Yaskawa INFORM job: SKRZYNIA_4040_0_STOPNI_1OBR.JBI

/JOB
//NAME SKRZYNIA_4040_0_STOPNI_1OBR
///FOLDERNAME 02-SKRZYNIE_JOBS
//POS
///NPOS 413,413,0,35,0,0
///TOOL 0
///POSTYPE PULSE
///PULSE
C00000=1055,-24125,84372,288,19725,204
C00001=1055,-24125,84372,288,19725,204
C00002=0,-15438,65714,0,-68532,0
C00003=25524,-25821,36823,19654,-58495,38520
C00004=23988,-24960,37134,18595,-57837,38812
C00005=22822,-23954,37534,17811,-57199,39017
C00006=22935,-24057,37491,17887,-57262,38997
C00007=20006,-24258,37408,15644,-56932,39751
C00008=24402,-25289,37013,18874,-58060,38740
C00009=22585,-24665,40358,17164,-59622,30036
C00010=23477,-23257,40205,18030,-58646,29630
C00011=22519,-22398,40568,17384,-58125,29795
C00012=22700,-22567,40495,17506,-58225,29764
C00013=19339,-22794,40398,14955,-57865,30607
C00014=24825,-24328,39798,18931,-59350,29401
C00015=32755,-32613,25711,29640,-48730,33694
C00016=25632,-30899,26166,23992,-46203,35378
C00017=24264,-29862,26497,22996,-45413,35639
C00018=24403,-29974,26459,23097,-45496,35612
C00019=20575,-30233,26374,19602,-44891,36810
C00020=26556,-31526,25988,24663,-46720,35206
C00021=31152,-34007,25432,27964,-49085,34371
C00022=14779,-22420,82153,5620,-31515,42478
C00023=14779,-22420,82153,5620,-31515,42478
C00024=27667,-31817,30876,40298,-29340,25942
C00025=30467,-34548,18624,42252,-31099,25545
C00026=27667,-31817,21023,40298,-29340,25942
C00027=26226,-30681,21430,39338,-28403,26129
C00028=26403,-30829,21375,39455,-28520,26106
C00029=23300,-31093,21277,35654,-27590,27434
C00030=27667,-31817,21023,40298,-29340,25942
C00031=33767,-35384,20030,44426,-32984,25136
C00032=17528,-33021,25719,14295,-44761,40001
C00033=28412,-21339,35361,20830,-70681,36412
C00034=27333,-20260,35973,20228,-70115,36596
C00035=27399,-20329,35933,20265,-70150,36584
C00036=24360,-20684,35731,18412,-69734,37326
C00037=28877,-18893,40191,20941,-72149,36569
C00038=27817,-32566,25782,25532,-47502,36865
C00039=25779,-31294,26110,24054,-46400,37243
C00040=24344,-30243,26427,23007,-45578,37515
C00041=24432,-30312,26405,23072,-45630,37498
C00042=20021,-30599,26315,19050,-44944,38872
C00043=26262,-31616,26021,24405,-46667,37153
C00044=27439,-32346,25835,25259,-47302,36935
C00045=25659,-31170,26146,23974,-46312,37260
C00046=24581,-30384,26384,23190,-45695,37464
C00047=24689,-30466,26358,23269,-45758,37444
C00048=20001,-30771,26264,18999,-45026,38899
C00049=26308,-31607,26026,24448,-46671,37139
C00050=26309,-31604,29506,24448,-46670,37138
///LIMIT ON
C00051=58801,-24999,56179,43319,-3155,35712
C00052=58801,-24999,56179,43319,-3155,35712
///LIMIT OFF
C00053=58801,-24999,56179,43319,-54497,35712
C00054=29920,-29398,24569,49034,-27892,27689
C00055=29115,-28721,24834,48649,-27358,27707
C00056=27674,-27540,25333,47889,-26423,27783
C00057=27794,-27645,25287,47952,-26502,27777
C00058=24751,-27949,25156,44290,-25406,29014
C00059=29115,-28721,24834,48649,-27358,27707
C00060=40370,-34602,23054,55084,-33911,26929
C00061=27585,-47842,-289,32095,-40789,28095
C00062=4801,-35772,25187,4593,-28023,-82032
C00063=17634,-23800,39238,9573,-31425,-73339
C00064=17634,-23800,39238,9573,-31425,-73339
C00065=16549,-22464,39800,8390,-30730,-72975
C00066=16684,-22641,39722,8536,-30818,-73021
C00067=16684,-19968,45512,8078,-32771,-72767
C00068=17634,-23800,39238,9573,-31425,-73339
C00069=17837,-21535,44509,9322,-33342,-73155
C00070=17837,-21535,44509,9322,-33342,-73155
C00071=16866,-20378,45014,8305,-32755,-72853
C00072=17032,-20588,44918,8481,-32857,-72905
C00073=17032,-17542,51480,8009,-35060,-72636
C00074=17837,-21535,44509,9322,-33342,-73155
C00075=-20829,-18800,50532,-12466,-37179,-77446
C00076=-19934,-17904,50946,-11618,-36715,-77676
C00077=-20044,-18019,50891,-11723,-36773,-77647
C00078=-20044,-15288,56753,-11218,-38713,-77950
C00079=-20966,-18928,50473,-12596,-37250,-77413
C00080=-20884,-26676,33664,-14451,-31668,-76336
C00081=-20884,-26676,33664,-14451,-31668,-76336
C00082=-19557,-25338,34176,-13080,-30873,-76751
C00083=-19691,-25483,34117,-13220,-30955,-76709
C00084=-19691,-22773,39998,-12506,-32911,-77106
C00085=-20642,-26447,33747,-14206,-31526,-76411
C00086=-33629,-40566,17444,-29603,-33447,-71192
C00087=-33629,-40566,17444,42578,-32312,-84654
C00088=-42160,-31266,16400,42578,-32312,-84654
C00089=-87798,-804,48829,-20188,-26072,-60966
C00090=-76454,-11934,10236,-25964,7954,-64922
C00091=-76448,-11928,10235,-25961,7944,-64914
C00092=-68643,-7759,-23318,-14097,50582,-74897
C00093=-70868,-8793,-8075,-29663,30364,-70765
C00094=-67243,-1968,12282,-49553,26687,-63567
C00095=-68655,-309,14069,-48513,25966,-64203
C00096=-67497,-1678,12591,-49367,26558,-63682
C00097=-71436,-723,2905,-26484,35140,-73726
C00098=-71436,176,6426,-27636,33595,-73066
C00099=-71434,778,8668,-28412,32633,-72624
C00100=-68624,-2689,-85,-28291,36551,-72622
C00101=-99375,3692,5712,40719,48607,-84097
C00102=-94964,4957,10918,40408,44640,-83792
C00103=-93063,6047,12199,39572,43744,-83178
C00104=-94964,4957,10918,40408,44640,-83792
C00105=-94964,5754,13918,41385,43553,-84439
C00106=-94964,4957,10918,40408,44640,-83792
C00107=-90271,-412,-5146,23417,46876,-76529
C00108=-83133,-4088,-8267,6704,41492,-71542
C00109=-83133,-4088,-8267,6704,41492,-71542
C00110=-83133,-4088,-8267,6704,41492,-11598
C00111=-83133,-16026,-8267,6704,41492,-11598
C00112=-83133,-16026,-8267,6704,41492,-11598
C00113=-48225,-19387,30619,3889,32460,-6728
C00114=56943,-39861,25115,1795,-37402,-69601
C00115=29960,-38386,-19607,-115769,-41858,-24264
C00116=65721,-6478,18155,-133323,-22195,3361
C00117=70544,4411,32968,-134868,-18623,4660
C00118=71874,8263,38598,-134556,-17327,4659
C00119=72629,9390,40002,-135279,-16924,5107
C00120=71441,7638,37831,-134139,-17555,4406
C00121=77146,8888,25050,-166574,-32612,18372
C00122=77146,10029,28643,-166204,-31014,18167
C00123=77146,11198,32202,-165803,-29459,17947
C00124=75508,4678,16951,-165715,-35157,17778
C00125=68680,12216,24468,-164340,-40455,-13359
C00126=68362,12845,25743,-164045,-40097,-13561
C00127=68362,13700,28585,-163752,-38808,-13742
C00128=68362,12845,25743,-164045,-40097,-13561
C00129=64993,-1168,28876,-102971,-10760,-49875
C00130=63888,481,30670,-102324,-11438,-50313
C00131=64993,-1168,28876,-102971,-10760,-49875
C00132=58588,-14653,4620,-120782,-19611,-35794
C00133=29960,-38386,-19607,-115769,-41858,-24264
C00134=56943,-39861,25115,1795,-37402,-69601
C00135=-1002,-39861,25115,1795,-37402,-69601
C00136=-1001,-39858,25114,1795,-37402,0
///LIMIT ON
C00137=6591,-33902,35532,5956,-1761,-1932
///LIMIT OFF
C00138=6592,-33900,35531,103508,-35512,-26314
C00139=-99253,-13690,44082,59847,13407,-31313
C00140=-85045,-36869,-4353,28502,-22832,-52282
C00141=-92346,-18713,13565,21110,-22545,-55257
C00142=-85732,-21202,11427,30682,-24763,-59235
C00143=-84559,-15616,15722,33768,-24118,-60665
C00144=-85817,-13999,17072,32355,-23435,-60109
C00145=-83260,-12880,18034,36130,-24218,-61709
C00146=-84150,-13282,17685,34842,-23935,-61163
C00147=-85365,-11775,19006,33430,-23307,-60600
C00148=-84150,-13282,17685,34842,-23935,-61163
C00149=-85786,-16909,14677,31743,-23900,-59790
C00150=-84150,-13282,17685,34842,-23935,-61163
C00151=-83215,-12861,18051,36194,-24233,-61735
C00152=-84150,-13282,17685,34842,-23935,-61163
C00153=-85327,-11825,18959,33476,-23327,-60618
C00154=-84150,-13282,17685,34842,-23935,-61163
C00155=-87841,-18519,13420,28367,-23534,-58339
C00156=-84150,-13282,17685,34842,-23935,-61163
C00157=-83292,-12894,18020,36083,-24208,-61688
C00158=-84150,-13282,17685,34842,-23935,-61163
C00159=-85185,-12008,18799,33646,-23400,-60687
C00160=-84150,-13282,17685,34842,-23935,-61163
C00161=-86371,-18277,13606,30568,-23951,-59265
C00162=-84345,-13370,17612,34554,-23873,-61041
C00163=-83240,-12871,18042,36158,-24225,-61720
C00164=-84345,-13370,17612,34554,-23873,-61041
C00165=-85365,-12110,18711,33368,-23345,-60568
C00166=-84345,-13370,17612,34554,-23873,-61041
C00167=-86191,-19647,12567,30467,-24278,-59187
C00168=-84345,-13372,17610,34552,-23873,-61039
C00169=-83096,-12807,18098,36363,-24268,-61804
C00170=-84345,-13372,17610,34552,-23873,-61039
C00171=-85268,-12232,18600,33480,-23393,-60612
C00172=-84345,-13372,17610,34552,-23873,-61039
C00173=-84814,-16043,15376,33312,-24093,-60464
C00174=-84104,-13265,17702,34906,-23948,-61189
C00175=-82960,-12743,18153,36555,-24313,-61887
C00176=-84104,-13265,17702,34906,-23948,-61189
C00177=-84979,-12194,18635,33901,-23496,-60788
C00178=-84104,-13265,17702,34906,-23948,-61189
C00179=-86610,-16845,14732,30573,-23614,-59301
C00180=-84104,-13265,17702,34906,-23948,-61189
C00181=-82793,-12667,18222,36790,-24370,-61986
C00182=-84104,-13265,17702,34906,-23948,-61189
C00183=-84888,-12305,18537,34004,-23540,-60830
C00184=-84104,-13265,17702,34906,-23948,-61189
C00185=-83806,-19585,12613,33764,-25080,-60559
C00186=-83675,-13072,17868,35530,-24083,-61453
C00187=-82553,-12556,18319,37130,-24451,-62127
C00188=-83675,-13072,17868,35530,-24083,-61453
C00189=-84378,-12223,18610,34735,-23716,-61138
C00190=-83675,-13072,17868,35530,-24083,-61453
C00191=-87149,-17993,13826,29513,-23647,-58830
C00192=-84104,-13265,17702,34906,-23948,-61189
C00193=-82640,-12594,18285,37014,-24425,-62079
C00194=-84104,-13265,17702,34906,-23948,-61189
C00195=-84792,-12429,18430,34119,-23592,-60877
C00196=-84104,-13265,17702,34906,-23948,-61189
C00197=-83583,-9185,30892,23668,-36042,-57025
C00198=-85789,-8328,35795,20592,-37093,-55378
C00199=-90262,-21765,2389,14114,-35574,-54847
C00200=-90262,-21765,2389,28730,-17672,-54847
C00201=-89967,-19086,25635,28730,-17672,-54847
C00202=568,-24029,84339,168,19981,112
C00203=568,-24677,83015,164,20405,113
C00204=101153,-24598,83176,165,20353,113
C00205=101153,-24598,83176,165,20353,113
C00206=87323,-6914,39851,-18853,-38149,44508
C00207=83118,-12818,18089,-36330,-24263,61791
C00208=81969,-12276,18566,-37944,-24648,62472
C00209=83118,-12818,18089,-36330,-24263,61791
C00210=83927,-11846,18941,-35423,-23842,61433
C00211=83118,-12818,18089,-36330,-24263,61791
C00212=83806,-19585,12613,-33764,-25080,60559
C00213=83148,-12832,18077,-36287,-24254,61773
C00214=81889,-12236,18598,-38058,-24676,62520
C00215=83148,-12832,18077,-36287,-24254,61773
C00216=83900,-11930,18867,-35446,-23862,61440
C00217=83148,-12832,18077,-36287,-24254,61773
C00218=86610,-16845,14732,-30573,-23614,59301
C00219=82493,-13239,17725,-37070,-24559,62089
C00220=81442,-12739,18159,-38529,-24915,62703
C00221=82493,-13239,17725,-37070,-24559,62089
C00222=83435,-12133,18689,-36040,-24063,61682
C00223=82493,-13239,17725,-37070,-24559,62089
C00224=84814,-16043,15376,-33312,-24093,60464
C00225=82555,-13613,17404,-36910,-24580,62015
C00226=81369,-13053,17885,-38558,-24979,62709
C00227=82555,-13613,17404,-36910,-24580,62015
C00228=83568,-12431,18429,-35805,-24046,61580
C00229=82555,-13613,17404,-36910,-24580,62015
C00230=86191,-19647,12567,-30467,-24278,59187
C00231=82500,-13648,17375,-36975,-24607,62039
C00232=81594,-13224,17740,-38236,-24911,62571
C00233=82500,-13648,17375,-36975,-24607,62039
C00234=83449,-12543,18332,-35941,-24104,61633
C00235=82500,-13648,17375,-36975,-24607,62039
C00236=86371,-18277,13606,-30568,-23951,59265
C00237=82904,-13790,17251,-36416,-24470,61808
C00238=81796,-13275,17692,-37971,-24838,62464
C00239=82904,-13790,17251,-36416,-24470,61808
C00240=83696,-12867,18046,-35547,-24051,61466
C00241=82904,-13790,17251,-36416,-24470,61808
C00242=87841,-18519,13420,-28367,-23534,58339
C00243=82748,-13879,17174,-36603,-24542,61883
C00244=81789,-13434,17554,-37946,-24861,62449
C00245=82748,-13879,17174,-36603,-24542,61883
C00246=83603,-12888,18026,-35668,-24086,61514
C00247=82748,-13879,17174,-36603,-24542,61883
C00248=85786,-16909,14677,-31743,-23900,59790
C00249=82339,-14116,16972,-37087,-24733,62079
C00250=81557,-13752,17280,-38171,-24994,62536
C00251=82339,-14116,16972,-37087,-24733,62079
C00252=83390,-12909,18006,-35951,-24172,61633
C00253=82339,-14116,16972,-37087,-24733,62079
C00254=85732,-21202,11427,-30682,-24763,59235
C00255=82398,-14365,16763,-36952,-24745,62014
C00256=81340,-13876,17176,-38416,-25096,62632
C00257=82398,-14365,16763,-36952,-24745,62014
C00258=83629,-12951,17972,-35620,-24090,61491
C00259=82398,-14365,16763,-36952,-24745,62014
C00260=83775,-36460,5778,-32556,-23750,56951
C00261=69856,-53931,-13446,-33557,-28911,29591
C00262=43695,-41610,22646,45477,-37580,9181
C00263=79833,-32060,29151,65065,-75499,17030
C00264=46589,-23543,32575,47437,-59456,19719
C00265=34343,-28703,20955,31522,-59937,26478
C00266=20601,-31966,9393,15671,-60680,34344
C00267=58029,-25484,23838,55879,-68285,17494
C00268=64424,-28491,31029,58630,-66351,17656
C00269=34280,-39622,35434,31197,-32089,9395
///LIMIT ON
C00270=0,-44757,54667,0,2744,0
C00271=16657,-42063,37160,20008,-15173,6616
///LIMIT OFF
C00272=40382,-38226,12225,48505,-40693,16039
C00273=55481,-27484,23768,62968,-54833,11978
C00274=49936,-26717,24128,59936,-52007,12579
C00275=40993,-34144,10907,45777,-50361,16414
C00276=55330,-33748,11238,57660,-59334,12681
C00277=78664,-24436,10378,82837,-79111,12029
C00278=75189,-23065,11287,81851,-76948,11927
C00279=75189,-45249,11287,81851,-38847,11927
C00280=39199,-45249,11287,81851,-83130,11927
C00281=39199,-45249,11287,81851,-83130,11927
C00282=0,-24026,84338,1,19977,2
C00283=0,-24026,84338,1,19977,2
C00284=4264,-34194,25387,4006,-26954,-29436
C00285=4264,-34194,25387,4006,-26954,-81856
C00286=-21478,-27798,32214,-15234,-31599,-76056
C00287=-19679,-23059,39354,-12567,-32689,-77067
C00288=-1354,-23265,40547,-1729,-32338,-75190
C00289=2474,-22926,41128,543,-32322,-74812
C00290=16724,-20576,44291,8212,-32395,-72836
C00291=21329,-26386,39716,13285,-34016,-74401
C00292=-23778,-26243,38799,-16502,-35132,-75964
C00293=-20075,-15782,55752,-11329,-38404,-77896
C00294=16874,-17447,51356,7863,-34895,-72604
C00295=18580,-28601,30698,11472,-29284,-74138
C00296=6126,-41331,18955,6697,-26557,-30383
C00297=1,-24024,84337,2,19973,1
C00298=-64243,-26178,31107,-39513,40312,-5844
C00299=-72148,3973,56008,-35470,42045,-10522
C00300=-72090,16396,76301,-42067,35650,-6519
C00301=-69388,15725,61378,-31740,35177,-8719
C00302=-69127,27099,75569,-32744,34250,-8088
C00303=-67573,2495,11285,-21767,57629,-15193
C00304=-77819,19629,29798,-10454,63174,-20704
C00305=-72990,23583,14304,-10735,77209,-20379
C00306=-74593,38003,46707,-11043,65751,-19814
C00307=-73236,38943,48295,-11400,65557,-19316
C00308=-73329,42107,51779,-6346,67443,-19636
C00309=-87142,34654,46174,17622,63862,-25393
C00310=-87240,36727,48611,18897,66604,-25032
C00311=-99033,21517,12213,24947,79702,-26203
C00312=-91500,-14196,-34781,24472,81625,-22832
C00313=-100472,-45007,-27818,8167,67201,-29302
C00314=0,-36642,16905,0,48372,0
C00315=66009,-61997,-62105,21406,63483,18379
C00316=97242,-23579,-39442,10179,68876,30321
C00317=73684,-7073,-17511,24638,68131,29022
C00318=59136,7235,6676,33270,66602,27507
C00319=54816,14937,6234,39741,69494,31070
C00320=54365,20668,19279,41017,66202,29418
C00321=64503,4223,2857,29650,48528,26647
C00322=75622,3202,-3149,3890,49494,34281
C00323=88036,13177,2413,-18568,66573,35876
C00324=90462,21593,10123,-22613,76266,34479
C00325=92450,29224,20002,-25750,81642,33727
C00326=94949,8131,-12163,-20291,74229,36861
C00327=94949,8084,-13484,-20215,75047,36712
C00328=70412,-34016,-52305,-11724,65624,29757
C00329=44268,-30306,-1568,-7370,48673,18708
C00330=1,-24024,84337,2,19973,1
C00331=1,-24024,84337,2,19973,1
C00332=35720,-26719,45333,36814,-39824,4350
C00333=31311,-24391,37012,30296,-51528,29736
C00334=34162,-17357,32183,27794,-74501,33367
C00335=48608,-25286,29226,41890,-68866,29453
C00336=62093,-26534,55494,45669,-73540,27410
C00337=1,-24024,84337,2,19973,1
C00338=39943,-41903,29008,37348,-30478,1122
C00339=50712,-45163,3694,54202,-48634,13777
C00340=33730,-38727,5060,44589,-38829,15717
C00341=40855,-40866,-13431,41867,-55631,22487
C00342=59329,-52422,-25741,69939,-52774,12149
C00343=61512,-31790,21528,108331,-82342,18812
C00344=13547,-32557,41617,75619,-64512,89
C00345=-91085,-34291,10385,1908,-24348,-42097
C00346=-86191,-19647,12567,30467,-24278,-59187
C00347=-99336,-11722,19052,-14323,-20229,-40037
C00348=-98356,-11562,19564,-10422,-20330,-41507
C00349=-99474,-20389,12397,-11593,-22150,-41069
C00350=0,-52280,40443,0,6876,0
C00351=98750,-34911,19055,13387,-20552,33529
C00352=85481,-22689,10385,-30594,-25183,59147
C00353=97204,-12655,18233,8807,-19987,42423
C00354=97248,-12883,18033,8874,-20029,42393
C00355=96230,-24528,9149,6144,-22576,43630
C00356=0,-52280,40443,0,6876,0
C00357=0,-27933,77061,0,20812,0
C00358=0,-27933,77061,0,20812,0
C00359=0,-52280,40443,0,6876,0
///LIMIT ON
C00360=-91970,-60791,14435,-3343,512,-9412
///LIMIT OFF
C00361=-99196,-15868,16098,-13748,-19297,-38710
C00362=-99196,-15868,16098,-13748,-19297,-38710
C00363=-99196,-15868,16098,-13748,-19297,-38710
C00364=-85896,-11794,19566,31613,-21074,-58206
C00365=-87494,-11929,19445,26784,-20178,-56163
C00366=-99562,-16264,15781,-14410,-19427,-38431
C00367=-99196,-15868,16098,-13748,-19297,-38710
///LIMIT ON
C00368=-91970,-60791,14435,-3343,512,-9412
///LIMIT OFF
C00369=0,-52280,40443,0,6876,0
///LIMIT ON
C00370=91083,-60784,14823,-9043,-825,15173
///LIMIT OFF
C00371=83869,-19403,12921,-33769,-24740,60260
C00372=83869,-19403,12921,-33769,-24740,60260
C00373=83420,-14897,16486,-35538,-24144,61113
C00374=90681,-11839,19658,-13770,-20778,51433
C00375=90505,-11641,19895,-14005,-20849,51502
C00376=95871,-14889,15992,4901,-19605,43825
C00377=83869,-19403,12921,-33769,-24740,60260
C00378=89829,-21430,11438,-24586,-23314,56383
C00379=568,-24029,84339,168,19981,112
///LIMIT ON
C00380=-91970,-60791,14435,-3343,512,-9412
///LIMIT OFF
C00381=-86948,-23217,10819,28314,-23349,-56438
C00382=-85895,-16522,15767,31843,-22281,-58087
C00383=-93744,1669,52928,2829,-38206,-34736
C00384=-93484,-766,47198,3260,-36104,-34933
C00385=-86145,-24679,9854,29028,-23971,-56682
///LIMIT ON
C00386=-100471,-58311,4157,14142,-4822,-27614
C00387=-68517,-58311,4157,14142,-4822,-27614
///LIMIT OFF
C00388=0,-52280,40443,0,6876,0
///LIMIT ON
C00389=91083,-60784,14823,-9043,-825,15173
///LIMIT OFF
C00390=83869,-19403,12921,-33769,-24740,60260
C00391=82620,-18743,14708,-32942,-26226,58979
C00392=84031,-4887,35984,-19530,-40379,54984
C00393=84316,-7987,27276,-19995,-38113,55712
C00394=84798,-22668,11879,-29033,-26372,57255
///LIMIT ON
C00395=91083,-60784,14823,-9043,-825,15173
///LIMIT OFF
C00396=0,-52280,40443,0,6876,0
C00397=-100896,-36216,1995,-16119,-20751,-34692
C00398=-97287,-29142,12714,-8673,-22288,-37832
C00399=-86191,-19647,12567,30467,-24278,-59187
C00400=-85671,-16302,15857,30808,-24404,-58999
C00401=-100216,-10426,22391,-15020,-22581,-38655
C00402=-96259,-10424,22189,-2878,-17380,-43087
C00403=-87910,-17792,15835,25414,-24996,-56048
C00404=-97287,-29142,12714,-8673,-22288,-37832
///LIMIT ON
C00405=0,-47400,49619,0,4231,0
///LIMIT OFF
C00406=92301,-25634,22749,2368,-15645,37646
C00407=83738,-18329,13570,-34202,-24868,60772
C00408=90255,-12942,18284,-15153,-20833,52586
C00409=93508,-13158,18002,-4292,-20124,47959
C00410=79675,-24852,9157,-38810,-28565,62243
C00411=91863,-41556,2664,1531,-13798,37970
///LIMIT ON
C00412=0,-46824,50714,0,3911,0
///LIMIT OFF
BC00000=320972
BC00001=320972
BC00002=320972
BC00003=320968
BC00004=320968
BC00005=320968
BC00006=320968
BC00007=320968
BC00008=320968
BC00009=382457
BC00010=382462
BC00011=382462
BC00012=382462
BC00013=382462
BC00014=382462
BC00015=430683
BC00016=430683
BC00017=430683
BC00018=430683
BC00019=430683
BC00020=430683
BC00021=430683
BC00022=339085
BC00023=401553
BC00024=461461
BC00025=458458
BC00026=461461
BC00027=461461
BC00028=461461
BC00029=461461
BC00030=461461
BC00031=461461
BC00032=594803
BC00033=620084
BC00034=620084
BC00035=620084
BC00036=620084
BC00037=620084
BC00038=616104
BC00039=616104
BC00040=616104
BC00041=616104
BC00042=616104
BC00043=616104
BC00044=662657
BC00045=662657
BC00046=662657
BC00047=662657
BC00048=662657
BC00049=662657
BC00050=641739
BC00051=560595
BC00052=677703
BC00053=677703
BC00054=696570
BC00055=696570
BC00056=696570
BC00057=696570
BC00058=696570
BC00059=696570
BC00060=696570
BC00061=796226
BC00062=742181
BC00063=757542
BC00064=757542
BC00065=757542
BC00066=757542
BC00067=757542
BC00068=757542
BC00069=761988
BC00070=761988
BC00071=761988
BC00072=761988
BC00073=761988
BC00074=761988
BC00075=761988
BC00076=761988
BC00077=761988
BC00078=761988
BC00079=761988
BC00080=761988
BC00081=761988
BC00082=761988
BC00083=761988
BC00084=761988
BC00085=761988
BC00086=761988
BC00087=761988
BC00088=761988
BC00089=761988
BC00090=761988
BC00091=779740
BC00092=790826
BC00093=807530
BC00094=807530
BC00095=807530
BC00096=807530
BC00097=807530
BC00098=807530
BC00099=807531
BC00100=807531
BC00101=807531
BC00102=807531
BC00103=807531
BC00104=807531
BC00105=807531
BC00106=807531
BC00107=797908
BC00108=783274
BC00109=758009
BC00110=758009
BC00111=758009
BC00112=724827
BC00113=690394
BC00114=761988
BC00115=761988
BC00116=761988
BC00117=778202
BC00118=783363
BC00119=783363
BC00120=783363
BC00121=783363
BC00122=783363
BC00123=783363
BC00124=783363
BC00125=783363
BC00126=783363
BC00127=783363
BC00128=783363
BC00129=783363
BC00130=783363
BC00131=783363
BC00132=777850
BC00133=731266
BC00134=700544
BC00135=700544
BC00136=761990
BC00137=692927
BC00138=692930
BC00139=692930
BC00140=762533
BC00141=794663
BC00142=810022
BC00143=810022
BC00144=810022
BC00145=810022
BC00146=810022
BC00147=810022
BC00148=810022
BC00149=748578
BC00150=748578
BC00151=748578
BC00152=748578
BC00153=748578
BC00154=748578
BC00155=687134
BC00156=687134
BC00157=687134
BC00158=687134
BC00159=687134
BC00160=687134
BC00161=625689
BC00162=625689
BC00163=625689
BC00164=625689
BC00165=625689
BC00166=625689
BC00167=564239
BC00168=564239
BC00169=564239
BC00170=564239
BC00171=564239
BC00172=564239
BC00173=502795
BC00174=502795
BC00175=502795
BC00176=502795
BC00177=502795
BC00178=502795
BC00179=441351
BC00180=441351
BC00181=441351
BC00182=441351
BC00183=441351
BC00184=441351
BC00185=379907
BC00186=379907
BC00187=379907
BC00188=379907
BC00189=379907
BC00190=379907
BC00191=318463
BC00192=318463
BC00193=318463
BC00194=318463
BC00195=318463
BC00196=318463
BC00197=318463
BC00198=349186
BC00199=336469
BC00200=336469
BC00201=336469
BC00202=336469
BC00203=511557
BC00204=512005
BC00205=363797
BC00206=318463
BC00207=319414
BC00208=319414
BC00209=319414
BC00210=319414
BC00211=319414
BC00212=379907
BC00213=380859
BC00214=380859
BC00215=380859
BC00216=380859
BC00217=380859
BC00218=441351
BC00219=442302
BC00220=442302
BC00221=442302
BC00222=442302
BC00223=442302
BC00224=502795
BC00225=502795
BC00226=502795
BC00227=502795
BC00228=502795
BC00229=502795
BC00230=564239
BC00231=565184
BC00232=565184
BC00233=565184
BC00234=565184
BC00235=565184
BC00236=625689
BC00237=626633
BC00238=626633
BC00239=626633
BC00240=626633
BC00241=626633
BC00242=687134
BC00243=688079
BC00244=688079
BC00245=688079
BC00246=688079
BC00247=688079
BC00248=748578
BC00249=749525
BC00250=749525
BC00251=749525
BC00252=749525
BC00253=749525
BC00254=810022
BC00255=810970
BC00256=810970
BC00257=810970
BC00258=810970
BC00259=810970
BC00260=774262
BC00261=650210
BC00262=631429
BC00263=625005
BC00264=625005
BC00265=624315
BC00266=623618
BC00267=623834
BC00268=635459
BC00269=570676
BC00270=385647
BC00271=351346
BC00272=383172
BC00273=364530
BC00274=364530
BC00275=325110
BC00276=325110
BC00277=401820
BC00278=422140
BC00279=393202
BC00280=393202
BC00281=494758
BC00282=543163
BC00283=635815
BC00284=723932
BC00285=729148
BC00286=761988
BC00287=761988
BC00288=759784
BC00289=759333
BC00290=757541
BC00291=751775
BC00292=747286
BC00293=761988
BC00294=761988
BC00295=761216
BC00296=764808
BC00297=612669
BC00298=628031
BC00299=628031
BC00300=684741
BC00301=704627
BC00302=729566
BC00303=761498
BC00304=761498
BC00305=789007
BC00306=789007
BC00307=789007
BC00308=789008
BC00309=789008
BC00310=789009
BC00311=789009
BC00312=789009
BC00313=703667
BC00314=662265
BC00315=745805
BC00316=784925
BC00317=784926
BC00318=784926
BC00319=815173
BC00320=815173
BC00321=815173
BC00322=815173
BC00323=815173
BC00324=815176
BC00325=815176
BC00326=815176
BC00327=788770
BC00328=788770
BC00329=719957
BC00330=597308
BC00331=473465
BC00332=476969
BC00333=487590
BC00334=487590
BC00335=487590
BC00336=494376
BC00337=636767
BC00338=698801
BC00339=743560
BC00340=743560
BC00341=743560
BC00342=743586
BC00343=743586
BC00344=611991
BC00345=615191
BC00346=564239
BC00347=564239
BC00348=625689
BC00349=625689
BC00350=544949
BC00351=570137
BC00352=565184
BC00353=565184
BC00354=626637
BC00355=626637
BC00356=541121
BC00357=608083
BC00358=454048
BC00359=454048
BC00360=454045
BC00361=454045
BC00362=314610
BC00363=314610
BC00364=314612
BC00365=376034
BC00366=376034
BC00367=454045
BC00368=454045
BC00369=454048
BC00370=454048
BC00371=415438
BC00372=318616
BC00373=318616
BC00374=318616
BC00375=380554
BC00376=380554
BC00377=415438
BC00378=495145
BC00379=373524
BC00380=454045
BC00381=498922
BC00382=498922
BC00383=498922
BC00384=438950
BC00385=437474
BC00386=437474
BC00387=437474
BC00388=437474
BC00389=454048
BC00390=497753
BC00391=503461
BC00392=517595
BC00393=463737
BC00394=442011
BC00395=454048
BC00396=437474
BC00397=673724
BC00398=673724
BC00399=685802
BC00400=686287
BC00401=687086
BC00402=740567
BC00403=748582
BC00404=637836
BC00405=521515
BC00406=621954
BC00407=688058
BC00408=688056
BC00409=749577
BC00410=749577
BC00411=627740
BC00412=538724
///POSTYPE BASE
///RECTAN
///RCONF 1,0,0,0,0,0,0,0,0,0,0,0,0,0,0,0,0,0,0,0,0,0,0,0
P00006=0.000,0.000,0.000,0.0000,0.0000,0.0000
///RCONF 0,0,0,0,0,0,0,0,0,0,0,0,0,0,0,0,0,0,0,0,0,0,0,0
P00021=6.550,-0.003,-5.735,0.0000,0.0000,0.0000
P00022=5.943,-0.018,-6.388,0.0000,0.0000,0.0000
P00023=7.025,-0.019,-7.168,0.0000,0.0000,0.0000
P00024=5.926,-0.047,-4.777,0.0000,0.0000,0.0000
///RCONF 1,0,0,0,0,0,0,0,0,0,0,0,0,0,0,0,0,0,0,0,0,0,0,0
P00100=-0.081,2.558,4.482,0.0000,0.0000,0.0000
P00101=0.030,-2.286,2.993,0.0000,0.0000,0.0000
P00102=-0.005,-1.108,1.644,0.0000,0.0000,0.0000
P00103=-0.094,-3.400,4.200,0.0000,0.0000,0.0000
P00104=0.043,-2.127,5.826,0.0000,0.0000,0.0000
P00105=-0.043,0.662,5.286,0.0000,0.0000,0.0000
P00106=-0.018,-2.519,0.237,0.0000,0.0000,0.0000
P00107=-0.008,-4.537,-4.500,0.0000,0.0000,0.0000
///RCONF 0,0,0,0,0,0,0,0,0,0,0,0,0,0,0,0,0,0,0,0,0,0,0,0
P00280=-0.761,-1.221,0.004,0.0000,0.0000,0.0000
///RCONF 1,0,0,0,0,0,0,0,0,0,0,0,0,0,0,0,0,0,0,0,0,0,0,0
P00281=-0.866,-3.587,-0.008,0.0000,0.0000,0.0000
///RCONF 0,0,0,0,1,0,0,0,0,0,0,0,0,0,0,0,0,0,0,0,0,0,0,0
P00290=-0.023,-0.050,5.560,0.0000,0.0000,0.0000
///RCONF 1,0,0,0,0,0,0,0,0,0,0,0,0,0,0,0,0,0,0,0,0,0,0,0
P00291=0.002,-0.893,4.526,0.0000,0.0000,0.0000
P00301=0.046,-2.112,7.779,0.0000,0.0000,0.0000
P00302=-0.180,-2.409,6.326,0.0000,0.0000,0.0000
///RCONF 0,0,0,0,0,0,0,0,0,0,0,0,0,0,0,0,0,0,0,0,0,0,0,0
P00303=-0.004,-1.437,-4.584,0.0000,0.0000,0.0000
P00304=0.028,-1.666,-4.234,0.0000,0.0000,0.0000
P00305=-0.003,-1.920,-3.501,0.0000,0.0000,0.0000
P00306=0.015,-2.252,-3.054,0.0000,0.0000,0.0000
P00307=0.019,-2.151,-5.077,0.0000,0.0000,0.0000
P00308=-0.003,-2.092,-4.888,0.0000,0.0000,0.0000
P00309=-0.040,-2.205,-4.992,0.0000,0.0000,0.0000
P00352=13.252,-0.027,-0.827,0.0000,0.0000,0.0000
P00353=10.971,-0.082,0.776,0.0000,0.0000,0.0000
P00354=-0.024,2.508,-1.824,0.0000,0.0000,0.0000
P00355=-0.001,2.528,-1.131,0.0000,0.0000,0.0000
P00356=-0.034,2.921,-0.262,0.0000,0.0000,0.0000
P00357=0.003,3.386,-0.091,0.0000,0.0000,0.0000
P00358=0.014,3.037,-0.020,0.0000,0.0000,0.0000
P00359=-0.005,2.731,0.912,0.0000,0.0000,0.0000
P00360=-0.011,3.412,0.438,0.0000,0.0000,0.0000
//INST
///DATE 2025/03/24 15:28
///ATTR SC,RW
///GROUP1 RB1,BS1
NOP
CALL JOB:MOVE_INTO_TUNNEL
MOVJ C00000 BC00000 VJ=30.00
'------------------------
'------------------------
'SPOINA SRODEK DOL
'------------------------
'------------------------
'POMIAR DO WYJ!! PRZEROBIC NA STD
MOVJ C00001 BC00001 VJ=40.00
MOVJ C00002 BC00002 VJ=40.00
SFTOF
'SPOINA_PODLOGA_BRAK_ROZP
'W3P
MOVJ C00003 BC00003 VJ=20.00 PL=0
MOVL C00004 BC00004 V=166.7 PL=0
REFP 3 C00005 BC00005
CALL JOB:SEARCH-R1
SET P0100 P0006
SFTON P0100
MOVL C00006 BC00006 V=66.7 PL=0
REFP 3 C00007 BC00007
CALL JOB:SEARCH-R1
SET P0100 P0006
SFTON P0100
MOVL C00008 BC00008 V=333.3 PL=0
SFTOF
'W3L
MOVL C00009 BC00009 V=666.7
MOVL C00010 BC00010 V=166.7 PL=0
REFP 3 C00011 BC00011
CALL JOB:SEARCH-R1
SET P0101 P0006
SFTON P0101
MOVL C00012 BC00012 V=166.7 PL=0
REFP 3 C00013 BC00013
CALL JOB:SEARCH-R1
SET P0101 P0006
SFTON P0101
MOVL C00014 BC00014 V=333.3 PL=0
SFTOF
'W9P
MOVL C00015 BC00015 V=666.7
MOVL C00016 BC00016 V=166.7
REFP 3 C00017 BC00017
CALL JOB:SEARCH-R1
SET P0102 P0006
SFTON P0102
MOVL C00018 BC00018 V=166.7 PL=0
REFP 3 C00019 BC00019
CALL JOB:SEARCH-R1
SET P0102 P0006
SFTON P0102
SFTOF
MOVL C00020 BC00020 V=333.3 PL=0
MOVJ C00021 BC00021 VJ=30.00
MOVJ C00022 BC00022 VJ=30.00
MOVJ C00023 BC00023 VJ=30.00
MOVJ C00024 BC00024 VJ=30.00
'W9L
MOVL C00025 BC00025 V=666.7
MOVL C00026 BC00026 V=166.7
REFP 3 C00027 BC00027
CALL JOB:SEARCH-R1
SET P0103 P0006
SFTON P0103
MOVL C00028 BC00028 V=166.7 PL=0
REFP 3 C00029 BC00029
CALL JOB:SEARCH-R1
SET P0103 P0006
SFTON P0103
MOVL C00030 BC00030 V=333.3 PL=0
SFTOF
MOVJ C00031 BC00031 VJ=30.00
'PRZEJAZ NAD BELKA
'W1P
SFTOF
MOVJ C00032 BC00032 VJ=20.00 PL=0
MOVL C00033 BC00033 V=166.7 PL=0
REFP 3 C00034 BC00034
CALL JOB:SEARCH-R1
SET P0104 P0006
SFTON P0104
MOVL C00035 BC00035 V=166.7 PL=0
REFP 3 C00036 BC00036
CALL JOB:SEARCH-R1
SET P0104 P0006
SFTON P0104
MOVL C00037 BC00037 V=333.3 PL=0
SFTOF
'W1L
MOVL C00038 BC00038 V=666.7
MOVL C00039 BC00039 V=166.7 PL=0
REFP 3 C00040 BC00040
CALL JOB:SEARCH-R1
SET P0105 P0006
SFTON P0105
MOVL C00041 BC00041 V=166.7 PL=0
REFP 3 C00042 BC00042
CALL JOB:SEARCH-R1
SET P0105 P0006
SFTON P0105
MOVL C00043 BC00043 V=333.3 PL=0
SFTOF
MOVL C00044 BC00044 V=666.7
'W10P
MOVL C00045 BC00045 V=166.7 PL=0
REFP 3 C00046 BC00046
CALL JOB:SEARCH-R1
SET P0106 P0006
SFTON P0106
MOVL C00047 BC00047 V=166.7 PL=0
REFP 3 C00048 BC00048
CALL JOB:SEARCH-R1
SET P0106 P0006
SFTON P0106
MOVL C00049 BC00049 V=333.3 PL=0
SFTOF
'W10L
MOVJ C00050 BC00050 VJ=30.00
MOVJ C00051 BC00051 VJ=30.00
MOVJ C00052 BC00052 VJ=30.00
MOVJ C00053 BC00053 VJ=30.00
MOVL C00054 BC00054 V=333.3
MOVL C00055 BC00055 V=166.7 PL=0
REFP 3 C00056 BC00056
CALL JOB:SEARCH-R1
SET P0107 P0006
SFTON P0107
MOVL C00057 BC00057 V=166.7 PL=0
REFP 3 C00058 BC00058
CALL JOB:SEARCH-R1
SET P0107 P0006
SFTON P0107
MOVL C00059 BC00059 V=333.3 PL=0
SFTOF
MOVJ C00060 BC00060 VJ=30.00
'PRZEJAZD
'POMIAR DO WYJ!! PRZEROBIC NA STD
'KONIEC
MOVJ C00061 BC00061 VJ=25.00
MOVJ C00062 BC00062 VJ=50.00
'W5L
MOVJ C00063 BC00063 VJ=30.00 PL=0
MOVL C00064 BC00064 V=166.7
REFP 3 C00065 BC00065
CALL JOB:SEARCH-R1
SET P0021 P0006
SFTON P0021
MOVL C00066 BC00066 V=166.7
REFP 3 C00067 BC00067
CALL JOB:SEARCH-R1
SET P0021 P0006
SFTON P0021
SFTOF
MOVL C00068 BC00068 V=166.7
'W6L
MOVJ C00069 BC00069 VJ=20.00 PL=0
MOVL C00070 BC00070 V=166.7
REFP 3 C00071 BC00071
CALL JOB:SEARCH-R1
SET P0022 P0006
SFTON P0022
MOVL C00072 BC00072 V=166.7
REFP 3 C00073 BC00073
CALL JOB:SEARCH-R1
SET P0022 P0006
SFTON P0022
SFTOF
MOVL C00074 BC00074 V=166.7
'W6P
MOVL C00075 BC00075 V=333.3 PL=0
REFP 3 C00076 BC00076
CALL JOB:SEARCH-R1
SET P0023 P0006
SFTON P0023
MOVL C00077 BC00077 V=166.7
REFP 3 C00078 BC00078
CALL JOB:SEARCH-R1
SET P0023 P0006
SFTON P0023
SFTOF
MOVL C00079 BC00079 V=166.7
'W5P
MOVJ C00080 BC00080 VJ=20.00 PL=0
MOVL C00081 BC00081 V=166.7
REFP 3 C00082 BC00082
CALL JOB:SEARCH-R1
SET P0024 P0006
SFTON P0024
MOVL C00083 BC00083 V=166.7
REFP 3 C00084 BC00084
CALL JOB:SEARCH-R1
SET P0024 P0006
SFTON P0024
SFTOF
MOVL C00085 BC00085 V=166.7
'W7A
MOVJ C00086 BC00086 VJ=40.00
MOVJ C00087 BC00087 VJ=40.00
MOVJ C00088 BC00088 VJ=40.00
MOVJ C00089 BC00089 VJ=40.00
MOVJ C00090 BC00090 VJ=40.00
MOVJ C00091 BC00091 VJ=40.00
MOVJ C00092 BC00092 VJ=40.00
MOVJ C00093 BC00093 VJ=40.00
MOVL C00094 BC00094 V=250.0
REFP 3 C00095 BC00095
CALL JOB:SEARCH-R1
SET P0280 P0006
SFTON P0280
MOVL C00096 BC00096 V=166.7
MOVL C00097 BC00097 V=250.0
MOVL C00098 BC00098 V=166.7
REFP 3 C00099 BC00099
CALL JOB:SEARCH-R1
SET P0280 P0006
MOVL C00100 BC00100 V=166.7
SFTOF
MOVL C00101 BC00101 V=333.3
MOVL C00102 BC00102 V=166.7
REFP 3 C00103 BC00103
CALL JOB:SEARCH-R1
SET P0290 P0006
SFTON P0290
MOVL C00104 BC00104 V=166.7
REFP 3 C00105 BC00105
CALL JOB:SEARCH-R1
SET P0290 P0006
MOVL C00106 BC00106 V=166.7
'DOKONCZYC SEARCH
'DOKONCZYC SEARCH
MOVJ C00107 BC00107 VJ=20.00
SFTOF
MOVJ C00108 BC00108 VJ=30.00
MOVJ C00109 BC00109 VJ=40.00
MOVJ C00110 BC00110 VJ=40.00
MOVJ C00111 BC00111 VJ=40.00
MOVJ C00112 BC00112 VJ=40.00
MOVJ C00113 BC00113 VJ=50.00
'W7B
MOVJ C00114 BC00114 VJ=50.00
MOVJ C00115 BC00115 VJ=50.00
MOVJ C00116 BC00116 VJ=30.00
MOVJ C00117 BC00117 VJ=20.00
MOVL C00118 BC00118 V=166.7
REFP 3 C00119 BC00119
CALL JOB:SEARCH-R1
SET P0281 P0006
MOVL C00120 BC00120 V=166.7
SFTON P0281
MOVL C00121 BC00121 V=166.7
MOVL C00122 BC00122 V=166.7
REFP 3 C00123 BC00123
CALL JOB:SEARCH-R1
SET P0281 P0006
MOVJ C00124 BC00124 VJ=15.00
SFTOF
MOVJ C00125 BC00125 VJ=20.00
MOVL C00126 BC00126 V=166.7
REFP 3 C00127 BC00127
CALL JOB:SEARCH-R1
SET P0291 P0006
MOVL C00128 BC00128 V=166.7
MOVL C00129 BC00129 V=166.7
REFP 3 C00130 BC00130
CALL JOB:SEARCH-R1
SET P0291 P0006
MOVL C00131 BC00131 V=166.7
MOVJ C00132 BC00132 VJ=30.00
MOVJ C00133 BC00133 VJ=30.00
MOVJ C00134 BC00134 VJ=50.00
MOVJ C00135 BC00135 VJ=50.00
'------------------------
'------------------------
'PRAWA STRONA PROFIL GORA
'------------------------
'------------------------
MOVJ C00136 BC00136 VJ=50.00
MOVJ C00137 BC00137 VJ=50.00
MOVJ C00138 BC00138 VJ=50.00
MOVJ C00139 BC00139 VJ=20.00
MOVJ C00140 BC00140 VJ=50.00
'------------------------
'W14A L
'------------------------
SFTOF
MOVJ C00141 BC00141 VJ=50.00
'------------------------
'W14A P
'------------------------
SFTOF
MOVJ C00142 BC00142 VJ=50.00
MOVJ C00143 BC00143 VJ=50.00
MOVL C00144 BC00144 V=166.7 PL=0
REFP 3 C00145 BC00145
CALL JOB:SEARCH-R1
SET P0301 P0006
SFTON P0301
MOVL C00146 BC00146 V=166.7 PL=0
REFP 3 C00147 BC00147
CALL JOB:SEARCH-R1
SET P0301 P0006
SFTON P0301
MOVL C00148 BC00148 V=166.7 PL=0
SFTOF
'------------------------
'W19A L
'------------------------
SFTOF
MOVJ C00149 BC00149 VJ=50.00
MOVL C00150 BC00150 V=200.0 PL=0
REFP 3 C00151 BC00151
CALL JOB:SEARCH-R1
SET P0302 P0006
SFTON P0302
MOVL C00152 BC00152 V=166.7 PL=0
REFP 3 C00153 BC00153
CALL JOB:SEARCH-R1
SET P0302 P0006
SFTON P0302
MOVL C00154 BC00154 V=250.0 PL=0
SFTOF
'------------------------
'W19A P
'------------------------
SFTOF
MOVJ C00155 BC00155 VJ=50.00
MOVL C00156 BC00156 V=166.7 PL=0
REFP 3 C00157 BC00157
CALL JOB:SEARCH-R1
SET P0303 P0006
SFTON P0303
MOVL C00158 BC00158 V=166.7 PL=0
REFP 3 C00159 BC00159
CALL JOB:SEARCH-R1
SET P0303 P0006
SFTON P0303
MOVL C00160 BC00160 V=166.7 PL=0
SFTOF
'------------------------
'W13A L
'------------------------
SFTOF
MOVJ C00161 BC00161 VJ=50.00
MOVL C00162 BC00162 V=166.7 PL=0
REFP 3 C00163 BC00163
CALL JOB:SEARCH-R1
SET P0304 P0006
SFTON P0304
MOVL C00164 BC00164 V=166.7 PL=0
REFP 3 C00165 BC00165
CALL JOB:SEARCH-R1
SET P0304 P0006
SFTON P0304
MOVL C00166 BC00166 V=166.7 PL=0
SFTOF
'------------------------
'W13A P
'------------------------
SFTOF
MOVJ C00167 BC00167 VJ=50.00
MOVL C00168 BC00168 V=200.0 PL=0
REFP 3 C00169 BC00169
CALL JOB:SEARCH-R1
SET P0305 P0006
SFTON P0305
MOVL C00170 BC00170 V=166.7 PL=0
REFP 3 C00171 BC00171
CALL JOB:SEARCH-R1
SET P0305 P0006
SFTON P0305
MOVL C00172 BC00172 V=250.0 PL=0
SFTOF
'------------------------
'W18A L
'------------------------
SFTOF
MOVJ C00173 BC00173 VJ=50.00
MOVL C00174 BC00174 V=200.0 PL=0
REFP 3 C00175 BC00175
CALL JOB:SEARCH-R1
SET P0306 P0006
SFTON P0306
MOVL C00176 BC00176 V=166.7 PL=0
REFP 3 C00177 BC00177
CALL JOB:SEARCH-R1
SET P0306 P0006
SFTON P0306
MOVL C00178 BC00178 V=166.7 PL=0
SFTOF
'------------------------
'W18A P
'------------------------
SFTOF
MOVJ C00179 BC00179 VJ=50.00
MOVL C00180 BC00180 V=200.0 PL=0
REFP 3 C00181 BC00181
CALL JOB:SEARCH-R1
SET P0307 P0006
SFTON P0307
MOVL C00182 BC00182 V=166.7 PL=0
REFP 3 C00183 BC00183
CALL JOB:SEARCH-R1
SET P0307 P0006
SFTON P0307
MOVL C00184 BC00184 V=166.7 PL=0
SFTOF
'------------------------
'W15A L
'------------------------
SFTOF
MOVJ C00185 BC00185 VJ=50.00
MOVL C00186 BC00186 V=200.0 PL=0
REFP 3 C00187 BC00187
CALL JOB:SEARCH-R1
SET P0308 P0006
SFTON P0308
MOVL C00188 BC00188 V=166.7 PL=0
REFP 3 C00189 BC00189
CALL JOB:SEARCH-R1
SET P0308 P0006
SFTON P0308
MOVL C00190 BC00190 V=166.7 PL=0
SFTOF
'------------------------
'W15A P
'------------------------
SFTOF
MOVJ C00191 BC00191 VJ=50.00
MOVL C00192 BC00192 V=166.7 PL=0
REFP 3 C00193 BC00193
CALL JOB:SEARCH-R1
SET P0309 P0006
SFTON P0309
MOVL C00194 BC00194 V=166.7 PL=0
REFP 3 C00195 BC00195
CALL JOB:SEARCH-R1
SET P0309 P0006
SFTON P0309
MOVL C00196 BC00196 V=166.7 PL=0
SFTOF
MOVL C00197 BC00197 V=333.3
'------------------------
'W17A L
'------------------------
MOVL C00198 BC00198 V=500.0
SFTOF
MOVJ C00199 BC00199 VJ=10.00
MOVJ C00200 BC00200 VJ=20.00
MOVJ C00201 BC00201 VJ=50.00
MOVJ C00202 BC00202 VJ=50.00
MOVJ C00203 BC00203 VJ=70.00
MOVJ C00204 BC00204 VJ=30.00
MOVJ C00205 BC00205 VJ=30.00
'------------------------
'------------------------
'LEWA STRONA PROFIL GORA
'------------------------
'------------------------
SFTOF
'POPRAWID DOJAZD
'------------------------
'W15B L
'------------------------
SFTOF
MOVJ C00206 BC00206 VJ=10.00
MOVL C00207 BC00207 V=166.7 PL=0
REFP 3 C00208 BC00208
CALL JOB:SEARCH-R1
SET P0352 P0006
SFTON P0352
MOVL C00209 BC00209 V=166.7 PL=0
REFP 3 C00210 BC00210
CALL JOB:SEARCH-R1
SET P0352 P0006
SFTON P0352
MOVL C00211 BC00211 V=166.7 PL=0
SFTOF
'------------------------
'W15B P
'------------------------
SFTOF
MOVJ C00212 BC00212 VJ=20.00
MOVL C00213 BC00213 V=166.7 PL=0
REFP 3 C00214 BC00214
CALL JOB:SEARCH-R1
SET P0353 P0006
SFTON P0353
MOVL C00215 BC00215 V=166.7 PL=0
REFP 3 C00216 BC00216
CALL JOB:SEARCH-R1
SET P0353 P0006
SFTON P0353
MOVL C00217 BC00217 V=166.7 PL=0
SFTOF
'------------------------
'W18B L
'------------------------
SFTOF
MOVJ C00218 BC00218 VJ=50.00
MOVL C00219 BC00219 V=166.7 PL=0
REFP 3 C00220 BC00220
CALL JOB:SEARCH-R1
SET P0354 P0006
SFTON P0354
MOVL C00221 BC00221 V=166.7 PL=0
REFP 3 C00222 BC00222
CALL JOB:SEARCH-R1
SET P0354 P0006
SFTON P0354
MOVL C00223 BC00223 V=166.7 PL=0
SFTOF
'------------------------
'W18B P
'------------------------
SFTOF
MOVJ C00224 BC00224 VJ=50.00
MOVL C00225 BC00225 V=166.7 PL=0
REFP 3 C00226 BC00226
CALL JOB:SEARCH-R1
SET P0355 P0006
SFTON P0355
MOVL C00227 BC00227 V=166.7 PL=0
REFP 3 C00228 BC00228
CALL JOB:SEARCH-R1
SET P0355 P0006
SFTON P0355
MOVL C00229 BC00229 V=166.7 PL=0
SFTOF
'------------------------
'W13B L
'------------------------
SFTOF
MOVJ C00230 BC00230 VJ=50.00
MOVL C00231 BC00231 V=166.7 PL=0
REFP 3 C00232 BC00232
CALL JOB:SEARCH-R1
SET P0356 P0006
SFTON P0356
MOVL C00233 BC00233 V=166.7 PL=0
REFP 3 C00234 BC00234
CALL JOB:SEARCH-R1
SET P0356 P0006
SFTON P0356
MOVL C00235 BC00235 V=166.7 PL=0
SFTOF
'------------------------
'W13B P
'------------------------
SFTOF
MOVJ C00236 BC00236 VJ=50.00
MOVL C00237 BC00237 V=166.7 PL=0
REFP 3 C00238 BC00238
CALL JOB:SEARCH-R1
SET P0357 P0006
SFTON P0357
MOVL C00239 BC00239 V=166.7 PL=0
REFP 3 C00240 BC00240
CALL JOB:SEARCH-R1
SET P0357 P0006
SFTON P0357
MOVL C00241 BC00241 V=166.7 PL=0
SFTOF
'------------------------
'W19B L
'------------------------
SFTOF
MOVJ C00242 BC00242 VJ=50.00
MOVL C00243 BC00243 V=166.7 PL=0
REFP 3 C00244 BC00244
CALL JOB:SEARCH-R1
SET P0358 P0006
SFTON P0358
MOVL C00245 BC00245 V=166.7 PL=0
REFP 3 C00246 BC00246
CALL JOB:SEARCH-R1
SET P0358 P0006
SFTON P0358
MOVL C00247 BC00247 V=166.7 PL=0
SFTOF
'------------------------
'W19B P
'------------------------
SFTOF
MOVJ C00248 BC00248 VJ=50.00
MOVL C00249 BC00249 V=166.7 PL=0
REFP 3 C00250 BC00250
CALL JOB:SEARCH-R1
SET P0359 P0006
SFTON P0359
MOVL C00251 BC00251 V=166.7 PL=0
REFP 3 C00252 BC00252
CALL JOB:SEARCH-R1
SET P0359 P0006
SFTON P0359
MOVL C00253 BC00253 V=166.7 PL=0
SFTOF
'------------------------
'W14B L
'------------------------
SFTOF
MOVJ C00254 BC00254 VJ=50.00
MOVL C00255 BC00255 V=166.7 PL=0
REFP 3 C00256 BC00256
CALL JOB:SEARCH-R1
SET P0360 P0006
SFTON P0360
MOVL C00257 BC00257 V=166.7 PL=0
REFP 3 C00258 BC00258
CALL JOB:SEARCH-R1
SET P0360 P0006
SFTON P0360
MOVL C00259 BC00259 V=166.7 PL=0
SFTOF
'------------------------
'W14B P
'------------------------
SFTOF
SFTOF
MOVJ C00260 BC00260 VJ=50.00
MOVJ C00261 BC00261 VJ=50.00
MOVJ C00262 BC00262 VJ=40.00
MOVL C00263 BC00263 V=166.7
SFTON P0105
MOVL C00264 BC00264 V=166.7
MACRO1 MJ#(0) ARGF24
ARCON
SFTON P0104
MOVL C00265 BC00265 V=11.3
MOVL C00266 BC00266 V=11.3
ARCOF
SFTOF
MOVL C00267 BC00267 V=333.3
MOVJ C00268 BC00268 VJ=20.00
MOVJ C00269 BC00269 VJ=30.00
MOVJ C00270 BC00270 VJ=70.00
MOVJ C00271 BC00271 VJ=30.00
MOVJ C00272 BC00272 VJ=20.00
MOVL C00273 BC00273 V=666.7
'**********************
'W3
'**********************
SFTON P0101
MOVL C00274 BC00274 V=166.7
ARCON
SFTON P0100
MOVL C00275 BC00275 V=11.7
ARCOF
MOVL C00276 BC00276 V=166.7
SFTOF
'SPOINA_PODLOGA_BRAK_ROZP
MOVJ C00277 BC00277 VJ=30.00
MOVJ C00278 BC00278 VJ=30.00
MOVJ C00279 BC00279 VJ=50.00
MOVJ C00280 BC00280 VJ=30.00
MOVJ C00281 BC00281 VJ=30.00
'**********************
'W5
'**********************
MOVJ C00282 BC00282 VJ=50.00
MOVJ C00283 BC00283 VJ=50.00
MOVJ C00284 BC00284 VJ=25.00
MOVJ C00285 BC00285 VJ=30.00
'**********************
'W5
MOVL C00286 BC00286 V=333.3
MACRO1 MJ#(0) ARGF9
SFTON P0024
MOVL C00287 BC00287 V=166.7
ARCON
WVON WEV#(2)
SFTON P0021
MOVL C00288 BC00288 V=9.2
WVON WEV#(3)
MOVL C00289 BC00289 V=9.2
WVON WEV#(2)
MOVL C00290 BC00290 V=9.2
ARCOF
WVOF
SFTOF
MOVJ C00291 BC00291 VJ=20.00
MOVJ C00292 BC00292 VJ=20.00
'**********************
'W6
'**********************
MACRO1 MJ#(0) ARGF9
SFTON P0023
MOVL C00293 BC00293 V=250.0
ARCON
WVON WEV#(2)
SFTON P0022
MOVL C00294 BC00294 V=9.2
ARCOF
WVOF
SFTOF
MOVJ C00295 BC00295 VJ=10.00
MOVJ C00296 BC00296 VJ=30.00
MOVJ C00297 BC00297 VJ=40.00
MOVJ C00298 BC00298 VJ=40.00
MOVJ C00299 BC00299 VJ=40.00
MOVJ C00300 BC00300 VJ=40.00
MOVJ C00301 BC00301 VJ=20.00
MOVJ C00302 BC00302 VJ=10.00
MOVJ C00303 BC00303 VJ=20.00
MOVL C00304 BC00304 V=166.7
MACRO1 MJ#(0) ARGF14
MOVL C00305 BC00305 V=166.7
SFTON P0280
MOVL C00306 BC00306 V=166.7 PL=0
ARCON ASF#(22)
MOVL C00307 BC00307 V=9.2
MOVL C00308 BC00308 V=9.2
SFTON P0290
MOVL C00309 BC00309 V=9.2
MOVL C00310 BC00310 V=9.2
ARCOF
SFTOF
MOVL C00311 BC00311 V=250.0
MOVL C00312 BC00312 V=416.7
MOVJ C00313 BC00313 VJ=30.00
MOVJ C00314 BC00314 VJ=30.00
MOVJ C00315 BC00315 VJ=30.00
MOVJ C00316 BC00316 VJ=30.00
MOVJ C00317 BC00317 VJ=30.00
'7b
MOVL C00318 BC00318 V=333.3
MOVL C00319 BC00319 V=333.3
SFTON P0281
MOVL C00320 BC00320 V=166.7 PL=0
ARCON ASF#(22)
MOVL C00321 BC00321 V=9.2
MOVL C00322 BC00322 V=9.2
SFTON P0291
MOVL C00323 BC00323 V=9.2
MOVL C00324 BC00324 V=9.2
MOVL C00325 BC00325 V=9.2
ARCOF
SFTOF
'TUTAJ DODAC 7
'TUTAJ DODAC 7
'TUTAJ DODAC 7
MOVL C00326 BC00326 V=333.3
MOVL C00327 BC00327 V=333.3
MOVL C00328 BC00328 V=333.3
MOVJ C00329 BC00329 VJ=20.00
MOVJ C00330 BC00330 VJ=30.00
MOVJ C00331 BC00331 VJ=50.00
MOVJ C00332 BC00332 VJ=50.00
'**********************
'W9
'**********************
MACRO1 MJ#(0) ARGF24
SFTON P0103
MOVL C00333 BC00333 V=250.0
ARCON
SFTON P0102
MOVL C00334 BC00334 V=10.8
ARCOF
SFTOF
MOVL C00335 BC00335 V=333.3
MOVJ C00336 BC00336 VJ=50.00
MOVJ C00337 BC00337 VJ=70.00
MOVJ C00338 BC00338 VJ=50.00
MOVJ C00339 BC00339 VJ=20.00
'**********************
'W10
'**********************
SFTON P0107
MOVL C00340 BC00340 V=250.0
ARCON
SFTON P0106
MOVL C00341 BC00341 V=11.3
ARCOF
SFTOF
MOVL C00342 BC00342 V=333.3
MOVJ C00343 BC00343 VJ=50.00
MOVJ C00344 BC00344 VJ=50.00
'**********************
'**********************
'POCZATEK SPAWANIA BOKI
'**********************
'**********************
MOVJ C00345 BC00345 VJ=50.00
MOVJ C00346 BC00346 VJ=50.00
'**********************
'W13A
'**********************
SFTON P0305
MOVL C00347 BC00347 V=250.0 PL=0
SFTOF
MACRO1 MJ#(0) ARGF10
ARCON
SFTON P0304
MOVL C00348 BC00348 V=10.8
ARCOF
SFTOF
MOVL C00349 BC00349 V=250.0
'W13B
MOVJ C00350 BC00350 VJ=30.00
MOVJ C00351 BC00351 VJ=50.00
MOVL C00352 BC00352 V=500.0
'**********************
'W13B
'**********************
SFTON P0356
MOVL C00353 BC00353 V=166.7 PL=0
SFTOF
ARCON
SFTON P0357
MOVL C00354 BC00354 V=10.8
ARCOF
SFTOF
MOVL C00355 BC00355 V=250.0
MOVJ C00356 BC00356 VJ=30.00
MOVJ C00357 BC00357 VJ=40.00
MOVJ C00358 BC00358 VJ=30.00
MOVJ C00359 BC00359 VJ=30.00
MOVJ C00360 BC00360 VJ=30.00
MOVJ C00361 BC00361 VJ=30.00
MOVJ C00362 BC00362 VJ=30.00
'**********************
'W15A
'**********************
SFTON P0309
MOVL C00363 BC00363 V=166.7
MOVL C00364 BC00364 V=166.7 PL=0
SFTOF
ARCON
SFTON P0308
MOVL C00365 BC00365 V=10.8
ARCOF
SFTOF
MOVL C00366 BC00366 V=150.0
MOVJ C00367 BC00367 VJ=30.00
MOVJ C00368 BC00368 VJ=50.00
MOVJ C00369 BC00369 VJ=50.00
MOVJ C00370 BC00370 VJ=50.00
MOVJ C00371 BC00371 VJ=50.00
MOVJ C00372 BC00372 VJ=50.00
'**********************
'W15B
'**********************
SFTON P0352
MOVL C00373 BC00373 V=250.0
MOVL C00374 BC00374 V=83.3 PL=0
SFTOF
ARCON
SFTON P0353
MOVL C00375 BC00375 V=10.8
ARCOF
MOVL C00376 BC00376 V=66.7
SFTOF
MOVJ C00377 BC00377 VJ=40.00
MOVJ C00378 BC00378 VJ=40.00
MOVJ C00379 BC00379 VJ=30.00
MOVJ C00380 BC00380 VJ=30.00
MOVJ C00381 BC00381 VJ=40.00
'**********************
'W18A
'**********************
SFTON P0306
MOVL C00382 BC00382 V=333.3
MOVL C00383 BC00383 V=166.7 PL=0
SFTOF
ARCON
SFTON P0307
MOVL C00384 BC00384 V=10.8
ARCOF
SFTOF
MOVL C00385 BC00385 V=250.0
MOVJ C00386 BC00386 VJ=30.00
MOVJ C00387 BC00387 VJ=30.00
MOVJ C00388 BC00388 VJ=50.00
MOVJ C00389 BC00389 VJ=50.00
MOVJ C00390 BC00390 VJ=50.00
'**********************
'W18B
'**********************
SFTON P0355
MOVL C00391 BC00391 V=166.7
MOVL C00392 BC00392 V=166.7 PL=0
SFTOF
ARCON
SFTON P0354
MOVL C00393 BC00393 V=10.8
ARCOF
MOVL C00394 BC00394 V=250.0
SFTOF
MOVJ C00395 BC00395 VJ=30.00
MOVJ C00396 BC00396 VJ=30.00
MOVJ C00397 BC00397 VJ=40.00
MOVJ C00398 BC00398 VJ=50.00
MOVJ C00399 BC00399 VJ=30.00
'**********************
'W19A
'**********************
MOVL C00400 BC00400 V=166.7
SFTON P0303
MOVL C00401 BC00401 V=166.7 PL=0
SFTOF
ARCON
SFTON P0302
MOVL C00402 BC00402 V=10.8
ARCOF
SFTOF
MOVL C00403 BC00403 V=150.0
MOVJ C00404 BC00404 VJ=30.00
MOVJ C00405 BC00405 VJ=50.00
MOVJ C00406 BC00406 VJ=50.00
'**********************
'W19B
'**********************
SFTON P0358
MOVL C00407 BC00407 V=500.0
MOVL C00408 BC00408 V=166.7 PL=0
SFTOF
ARCON
SFTON P0359
MOVL C00409 BC00409 V=10.8
ARCOF
SFTOF
MOVL C00410 BC00410 V=250.0
MOVJ C00411 BC00411 VJ=40.00
MOVJ C00412 BC00412 VJ=50.00
CALL JOB:MOVE_OUT_OF_TUNNEL
END
